TYPE E_TestWithNegatives :
(
	Negative := -1,
	Zero := 0,
	One := 1,
	MAX_E_TestWithNegatives
);
END_TYPE

(* stored: Version 1.1.0.1, ProductVersion 3.1.0.36
   DUT E_TestWithNegatives: Id {8e7aacb5-ce34-417e-bdc4-860d34bee96e} *)
